// Mitsubishi GX Works2 project: EX2_   PLC: FX3G

// global labels: Global1
VAR_GLOBAL
  CastingMachine AT M0 : BOOL;
  Lamp2 AT Y002 : BOOL;
  ErrorAtCast AT X006 : BOOL;
  Sen_60 AT X000 : BOOL;
  Sen_70 AT X001 : BOOL;
END_VAR
VAR_GLOBAL CONSTANT
  TenSecond : INT := 10;
END_VAR
VAR_GLOBAL
  CountingChairs AT CC1 : BOOL;
END_VAR
VAR_GLOBAL CONSTANT
  Two : INT := 2;
END_VAR
VAR_GLOBAL
  TwoHundred AT CS1 : BOOL;
  Sen_10 AT X005 : BOOL;
  Sen_20 AT X004 : BOOL;
  Lamp1 AT Y001 : BOOL;
  Switch10 AT X010 : BOOL;
  ChairReady AT X002 : BOOL;
  FinishCast AT M3 : BOOL;
END_VAR

// task Task_01 (event TRUE, interval 0, priority 31): POU_01

PROGRAM POU_01
VAR CONSTANT
  Sec : INT := 5;
END_VAR
(* structured ladder/FBD written out as ST: instructions are called as NAME(EN, inputs, outputs); _pN, _eN, _tN stand for wires *)
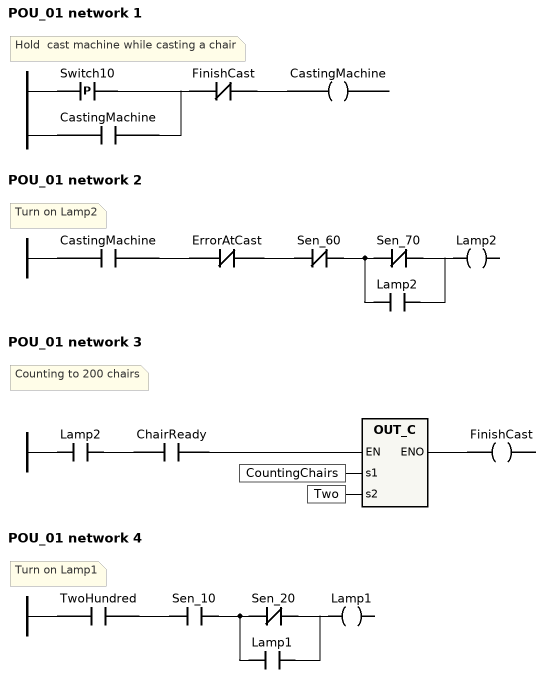
(* network 1 *)
(* Hold  cast machine while casting a chair *)
CastingMachine := (LDP(TRUE, Switch10) OR CastingMachine) AND NOT FinishCast;
(* network 2 *)
(* Turn on Lamp2 *)
_p1 := CastingMachine AND NOT ErrorAtCast AND NOT Sen_60;
Lamp2 := (_p1 AND NOT Sen_70) OR (_p1 AND Lamp2);
(* network 3 *)
(* Counting to 200 chairs *)
_e1 := OUT_C(Lamp2 AND ChairReady, CountingChairs, Two);
FinishCast := _e1;
(* network 4 *)
(* Turn on Lamp1 *)
_p1 := TwoHundred AND Sen_10;
Lamp1 := (_p1 AND NOT Sen_20) OR (_p1 AND Lamp1);
END_PROGRAM
